FUNCTION_BLOCK E_RS (* Event-driven bistable,Reset dominant *)
  (* Standard: 61499-1-A.1; Classification: Event Processing *)
  (* Version 0.1, 2001-08-16, JHC, Rockwell Automation, XML version *)
  (* Version 0.0, 1998-04-11, JHC, Rockwell Automation, SRC version *)
  (* Compiler header: package fb.rt.events; *)
  (* Compiler Java IBM VisualAge 3.0 *)
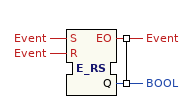
  EVENT_INPUT
    S; (* Set Event *)
    R; (* Reset Event *)
  END_EVENT
  EVENT_OUTPUT
    EO WITH Q; (* Output Event *)
  END_EVENT
  VAR_OUTPUT
    Q : BOOL; (* Current Output State *)
  END_VAR
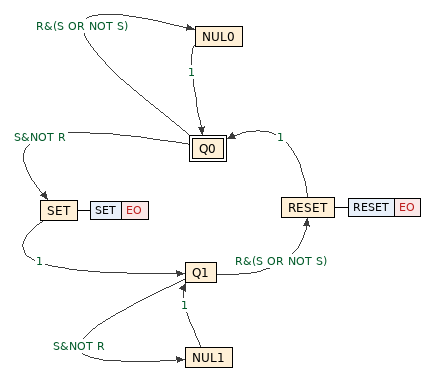
  EC_STATES
    Q0; (* Q is FALSE *)
    RESET : RESET -> EO; (* Reset Q and issue EO *)
    Q1; (* Q is TRUE *)
    NUL1; (* No action when Q is TRUE *)
    SET : SET -> EO; (* Set Q and issue EO *)
    NUL0; (* No action when Q is FALSE *)
  END_STATES
  EC_TRANSITIONS
    Q0 TO NUL0 := R&(S OR NOT S);
    NUL0 TO Q0 := 1;
    Q0 TO SET := S&NOT R;
    SET TO Q1 := 1;
    Q1 TO NUL1 := S&NOT R;
    NUL1 TO Q1 := 1;
    Q1 TO RESET := R&(S OR NOT S);
    RESET TO Q0 := 1;
  END_TRANSITIONS
  ALGORITHM SET IN ST: (* Set Q *)
Q:=TRUE;
  END_ALGORITHM
  ALGORITHM RESET IN ST: (* Reset Q *)
Q:=FALSE;
  END_ALGORITHM
END_FUNCTION_BLOCK
